PROGRAM ITCommunication
VAR_INPUT
	IbStartConnection:BOOL;
	IbPublishStart:BOOL;
END_VAR
VAR_OUTPUT
	QbOnline : BOOL;
END_VAR
VAR
	//Lit l'adresse IP de l'automate
	FB_MDP_NIC_Read    : FB_MDP_NIC_Read;
	iAddPoint		   : INT;
END_VAR

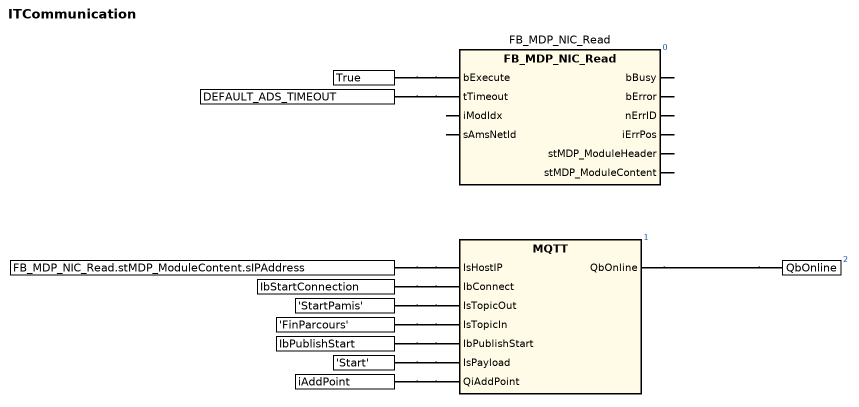
FB_MDP_NIC_Read(bExecute := True, tTimeout := DEFAULT_ADS_TIMEOUT);
MQTT(IsHostIP := FB_MDP_NIC_Read.stMDP_ModuleContent.sIPAddress, IbConnect := IbStartConnection, IsTopicOut := 'StartPamis', IsTopicIn := 'FinParcours', IbPublishStart := IbPublishStart, IsPayload := 'Start', QiAddPoint := iAddPoint);
QbOnline := MQTT.QbOnline;

END_PROGRAM

(* stored: Version 1.1.0.1, ProductVersion 3.1.4024.12
   POU ITCommunication: Id {5aa8df56-51b8-455f-8faa-b81449422817}, SpecialFunc None *)
